Omron CX-Programmer project NewProject (CX-Programmer 9.50)

# PLC projek_conveyer: CJ1M CPU11

## Global symbols (name address type ; comment)
0.01 BOOL  ; Kanan/Panjang

## Program NewProgram1 (cyclic task 0)
Local symbols
CNT 0.00 BOOL  ; 0.04
TIM 0.00 BOOL  ; timer 1 detik

### Section Section1

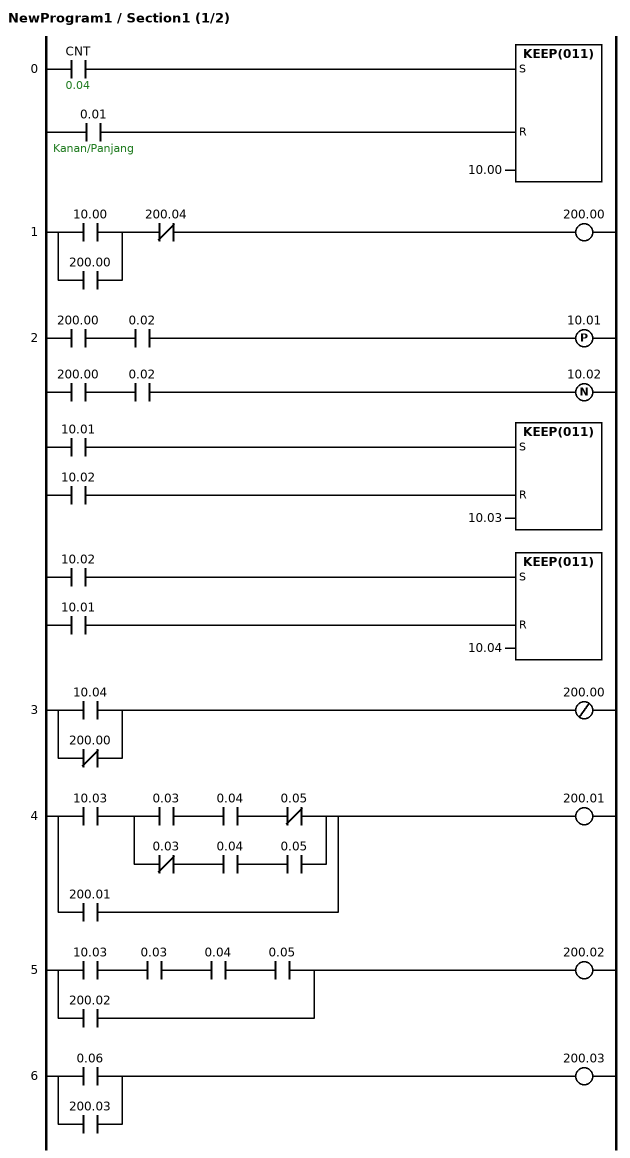
; rung 0
LD CNT  ; 0.04
LD 0.01  ; Kanan/Panjang
KEEP(011) 10.00
; rung 1
LD 10.00
OR 200.00
ANDNOT 200.04
OUT 200.00
; rung 2
LD 200.00
AND 0.02
DIFU(013) 10.01
LD 200.00
AND 0.02
DIFD(014) 10.02
LD 10.01
LD 10.02
KEEP(011) 10.03
LD 10.02
LD 10.01
KEEP(011) 10.04
; rung 3
LD 10.04
ORNOT 200.00
OUTNOT 200.00
; rung 4
LD 10.03
LD 0.03
AND 0.04
ANDNOT 0.05
LDNOT 0.03
AND 0.04
AND 0.05
ORLD
ANDLD
OR 200.01
OUT 200.01
; rung 5
LD 10.03
AND 0.03
AND 0.04
AND 0.05
OR 200.02
OUT 200.02
; rung 6
LD 0.06
OR 200.03
OUT 200.03

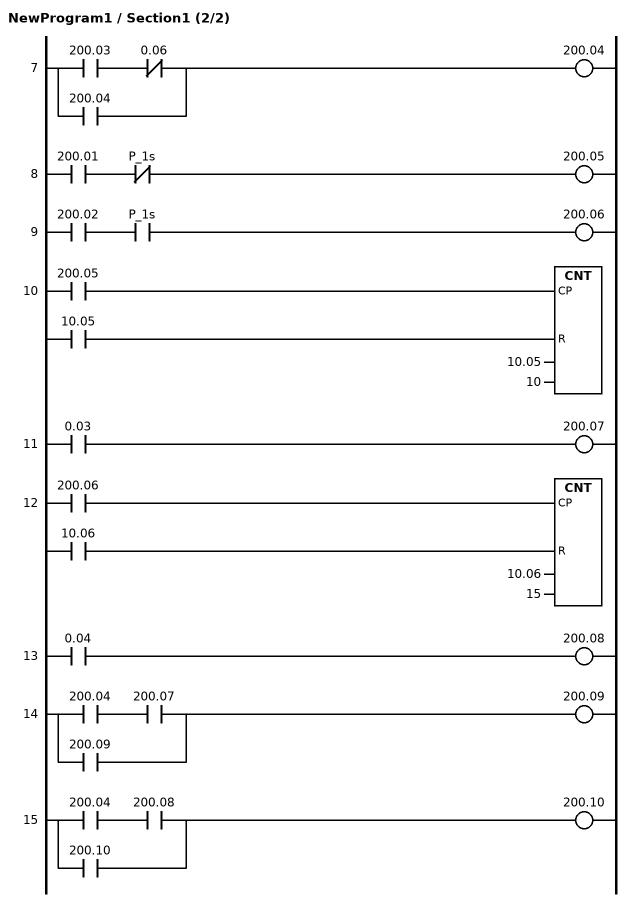
; rung 7
LD 200.03
ANDNOT 0.06
OR 200.04
OUT 200.04
; rung 8
LD 200.01
ANDNOT P_1s
OUT 200.05
; rung 9
LD 200.02
AND P_1s
OUT 200.06
; rung 10
LD 200.05
LD 10.05
CNT 10.05 10
; rung 11
LD 0.03
OUT 200.07
; rung 12
LD 200.06
LD 10.06
CNT 10.06 15
; rung 13
LD 0.04
OUT 200.08
; rung 14
LD 200.04
AND 200.07
OR 200.09
OUT 200.09
; rung 15
LD 200.04
AND 200.08
OR 200.10
OUT 200.10

### Section END
; rung 0
END(001)